{attribute 'qualified_only'}
{attribute 'strict'}
TYPE DropdownBox :
(
	first_page,
	Second_page
);
END_TYPE

(* stored: Version 1.1.0.1, ProductVersion 3.1.4024.12
   DUT DropdownBox: Id {679ade71-9d69-4fc8-9aa7-64b041b5ea35} *)
